Fanuc KAREL source: kf00105.KL

PROGRAM KF00105
%NOLOCKGROUP
%ENVIRONMENT REGOPE
VAR
I:INTEGER;J:INTEGER;X:REAL;Y:REAL;B:BOOLEAN;C:BOOLEAN;TXT : STRING[80];TXT2 : STRING[80];AI : ARRAY[4] OF INTEGER;BI : ARRAY[4] OF INTEGER;P : XYZWPR
JP : JOINTPOS9
PF : POSITION
V1 : VECTOR
V2 : VECTOR
STATUS:INTEGER
BEGIN
--
--
--
--
--
--
--
--
--
--
I=3
X=2.5
GET_REG_CMT(1,TXT,STATUS)
END KF00105
